(*
Sets the beam class assertion lines for a given beam class.
*)
FUNCTION_BLOCK FB_BeamClassOutputs
VAR_INPUT
	i_ArbiterBP	:	ST_BeamParams;
END_VAR
VAR_OUTPUT
END_VAR
VAR
	wBeamClass	:	BYTE;
	q_BC_ASSERTION_LINES	AT	%Q*	: ARRAY [0..15] OF	BOOL;
	InitCounter: INT;
END_VAR


//Beam Class
////////////////////////////////////
//0x0 = 0000 0000 0000 0000
//0xF = 1111 1111 1111 1111

//Initialize BC lines to zero on every pass
FOR InitCounter := 0 TO 15 DO
	q_BC_ASSERTION_LINES[InitCounter] := FALSE;
END_FOR

//Set BC lines according to beam class
FOR wBeamClass:=i_ArbiterBP.nBeamClass TO 0 BY -1 DO
	q_BC_ASSERTION_LINES[wBeamClass] := TRUE;
END_FOR

END_FUNCTION_BLOCK

(* stored: Version 1.1.0.1, ProductVersion 3.1.4022.12
   POU FB_BeamClassOutputs: Id {a28c1376-360b-0b96-3d68-05f53a5ce904}, SpecialFunc None *)
